# EPICS alarm handler configuration: alh_files/mgnt_li25_lgps.alhConfig
GROUP NULL LGPS:LI25:MG01
   $COMMAND edm -x -eolc -noedit mgnt_li25_lgps.edl
$ALIAS LGPS
$GUIDANCE
Li25 LGPS Magnets
   Group Name: LGPS:LI25:MG01
   Summary PV:  LGPS:LI25:MG01:STATSUMY
$END

GROUP LGPS:LI25:MG01  LGPS:LI25:2
   $COMMAND edm -x -eolc -noedit -m "DEV=LGPS:LI25:2" mgnt_unit.edl
CHANNEL   LGPS:LI25:2       LGPS:LI25:2:STATMSG                 -----
   $FORCEPV LGPS:LI25:2:STATMSGSV -DATL 1 0
